FUNCTION F_GetTimeSinceLastExternalTrigger : LREAL // [us]
VAR_INPUT
    LastExternalTriggerTimeLatch : ULINT; // [ns]
END_VAR
VAR
    dcSysTime : ULINT; // [ns]
END_VAR


dcSysTime := F_GetCurDcTickTime64();

IF dcSysTime > LastExternalTriggerTimeLatch THEN
    F_GetTimeSinceLastExternalTrigger := ULINT_TO_LREAL(dcSysTime - LastExternalTriggerTimeLatch) / 1000.0;
ELSE
    F_GetTimeSinceLastExternalTrigger := -ULINT_TO_LREAL(LastExternalTriggerTimeLatch - dcSysTime) / 1000.0;
END_IF

END_FUNCTION

(* stored: Version 1.1.0.1
   POU F_GetTimeSinceLastExternalTrigger: Id {dc0510a9-3904-4051-87f0-e9d882ae1b57}, SpecialFunc None *)
